(* PLC project  *)

PROGRAM A

bare text, which does not validate
END_PROGRAM
